(* CoDeSys 2.3 export: EXTOUTST.EXP *)

(* Data type in BathFB *)
(*Дополнительные выходы ванны*)
TYPE ExtOutST :
STRUCT
    remTime:     TIME;    (*оставшееся время*)
    bathEmpty:   BOOL;    (*ванна пуста*)
END_STRUCT
END_TYPE
